TYPE strQueueDetailExtended EXTENDS strQueueDetail :
	STRUCT
		aDATA			: ARRAY [0..Sewts_TCP.MAX_QueueData] OF BYTE ;	(* Data *)
	END_STRUCT
END_TYPE

(* stored: Version 1.1.0.1, ProductVersion 3.1.4024.12
   DUT strQueueDetailExtended: Id {4ff60372-d25d-4f70-9dc7-20c4488c3682} *)
